FUNCTION derivcvar_M_HardwareMap_t: LREAL
VAR_INPUT
    state: STATE;
END_VAR

derivcvar_M_HardwareMap_t := 1.0;

END_FUNCTION

(* stored: Version 1.1.0.1, ProductVersion 3.1.4022.18
   POU derivcvar_M_HardwareMap_t: Id {65c73318-e044-4b06-aed0-7f695df5f7d3}, SpecialFunc None *)
